// TIA Portal V16 export
// export: Created 2021-06-28T11:45:27.8781745Z, ExportSetting WithDefaults, DisplayName Totally Integrated Automation Portal, DisplayVersion V16 Update 4, DisplayName TIA Portal Version Control Interface, DisplayVersion V16 Update 2, DisplayName TIA Portal Openness, DisplayVersion V16 Update 4, DisplayName STEP 7 Professional, DisplayVersion V16 Update 4, DisplayName STEP 7 Safety, DisplayVersion V16, DisplayName WinCC Advanced, DisplayVersion V16 Update 4
FUNCTION "MQTT_MESSAGES_SEND" : Void   // FC10, FBD
{ S7_Optimized_Access := 'TRUE' }
VERSION : 0.1
// MQTT MESSAGES
// stored: AutoNumber true, IsIECCheckEnabled false, SetENOAutomatically false, UDAEnableTagReadback false
   VAR_TEMP
      TEMP0 : String;
      TEMP1 : String;
      TEMP3 : String;
      TEMP4 : String;
      TEMP5 : String;
      TEMP11 : String;
      wtemp1 : WString;
      wtemp2 : WString;
      wtemp3 : WString;
      wtemp4 : WString;
      TEMP6 : String;
      temp13 : String;
      temp14 : String;
      temp15 : String;
      wtemp14 : WString;
      wtemp16 : WString;
      temp110 : String;
      wtemp_null : WString;
      temp_rej1 : String;
      temp_rej2 : WString;
      TEMP : WString;
      TEMP_REJECT_TM_STMP : String;
      TEMP_BIT_BOOL1 : Bool;
   END_VAR
BEGIN

REGION Network 1 (SCL): Message_UID
   // MESSAGE_UID_FORMAT
   "MQTT_BLOCK".MSG_UID_data := CONCAT(IN1 := '"', IN2 :="MQTT_BLOCK".INDUCT_ID, IN3 := '_', IN4 := "MQTT_BLOCK".TIMESTAMP, IN5 := '"');
END_REGION

REGION Network 2 (SCL): CommonMessage
   // COMMON_MESSAGE
   "MQTT_BLOCK".COMMON_MESSAGE:=CONCAT(IN1:='{"message_uid":',IN2:="MQTT_BLOCK".MSG_UID_data,IN3:=',"induct_id":',IN4:="MQTT_BLOCK".INDUCT_ID,IN5:=',"timestamp":',
                                       IN6:="MQTT_BLOCK".TIMESTAMP,IN7:=',"data":{');
END_REGION

REGION Network 3 (SCL): ShipmentInfoMessage_ok_28.3.2021
   // // shipment INFO MQTT Message//
   IF "Info_Time_Mov_Bit" THEN
       #TEMP1 := CONCAT(IN1 := '{"message_uid":', IN2 := '"', IN3 := "MQTT_BLOCK".INDUCT_ID, IN4 := '_', IN5 := "MQTT_BLOCK".TimeStamp_Info, IN6 := '","induct_id":', IN7 := "MQTT_BLOCK".INDUCT_ID, IN8 := ',"timestamp":', IN9 := "MQTT_BLOCK".TimeStamp_Info, IN10 := ',"data":{"weight":', IN11 := "DATA_TCP".weight_string, IN12 := ',"barcodes":[');
       #TEMP3 := CONCAT(IN1 := '],"height":', IN2 := "DATA_TCP".STRING_H_INFO, IN3 := ',"length":', IN4 := "DATA_TCP".STRING_L_INFO, IN5 := ',"breadth":', IN6 := "DATA_TCP".STRING_B_INFO, IN7 := ',"weight_status_code":"',
                        IN8 := "MQTT_BLOCK".WEIGHT_STATUS_CODE, IN9 := '","vms_status_code":"', IN10 := "MQTT_BLOCK".VMS_STATUS_CODE, IN11 := '","scan_status_code":"',
                        IN12 := "MQTT_BLOCK".SCAN_STATUS_CODE, IN13 := '","uid":', IN14 := "MQTT_BLOCK".uid_1, IN15 := '');
       #wtemp1 := STRING_TO_WSTRING(#TEMP1);
       #wtemp4 := STRING_TO_WSTRING("DATA_TCP".String_To_String_Barcode);

       #wtemp2 := STRING_TO_WSTRING(#TEMP3);
       #wtemp3 := STRING_TO_WSTRING('}}');

       IF "DATA_TCP".STRING_L = '' THEN
           "DATA_TCP".STRING_L_INFO := '0';
       ELSE
           "DATA_TCP".STRING_L_INFO := "DATA_TCP".STRING_L;
       END_IF;

       IF "DATA_TCP".STRING_B = '' THEN
           "DATA_TCP".STRING_B_INFO := '0';
       ELSE
           "DATA_TCP".STRING_B_INFO := "DATA_TCP".STRING_B;
       END_IF;
       IF "DATA_TCP".STRING_H = '' THEN
           "DATA_TCP".STRING_H_INFO := '0';
       ELSE
           "DATA_TCP".STRING_H_INFO := "DATA_TCP".STRING_H;
       END_IF;


       IF "Aligner_Buffer_Module_Status" = 20 THEN
           "MQTT_BLOCK".MQTT_SHIPMENT_INFO := #wtemp_null;

       ELSIF "Aligner_Buffer_Module_Status" <> 20 & "Aligner_Buffer_Module_Status" < 300 THEN
           "MQTT_BLOCK".MQTT_SHIPMENT_INFO := CONCAT_WSTRING(IN1 := #wtemp1, IN2 := #wtemp4, IN3 := #wtemp2, IN4 := #wtemp3);
       END_IF;
       IF #wtemp4 = STRING_TO_WSTRING("DATA_TCP".String_To_String_Barcode) THEN
           "Trig_Info_CMD" := 1;
       END_IF;
       END_IF;
   // program end for shipment_info//
END_REGION

REGION Network 4 (SCL): HealthMessage WITH ERROR CODES
   // Induct Health MQTT Message
   IF "TIME_MOVE_HEALTH" & "ActualHealthStatus"=0 THEN
       IF "MQTT_BLOCK"."MQTT-OK" = 0 THEN "MQTT_BLOCK".health_induct_mqtt.message := '1'; "HEALTH_TR_2" := 1;
       ELSIF "Function_DB".IN_DWS_Alarm_DB = 0 THEN "MQTT_BLOCK".health_induct_mqtt.message := '403'; "HEALTH_TR_2" := 1;
       ELSIF "Function_DB".IN_Aligner_Alarm_DB  THEN "MQTT_BLOCK".health_induct_mqtt.message := '401'; "HEALTH_TR_2" := 1;
       ELSIF "Function_DB".IN_Barrier_Alarm_DB = 0 THEN "MQTT_BLOCK".health_induct_mqtt.message := '407'; "HEALTH_TR_2" := 1;
       ELSIF "Function_DB".IN_BUFFER_LEFT_ALARM_DB = 0 THEN "MQTT_BLOCK".health_induct_mqtt.message := '408'; "HEALTH_TR_2" := 1;
       ELSIF "Function_DB".IN_Buffer_Right_Alarm_DB = 0 THEN "MQTT_BLOCK".health_induct_mqtt.message := '409'; "HEALTH_TR_2" := 1;
       ELSIF "Error_Bit_Weight_Module"  THEN "MQTT_BLOCK".health_induct_mqtt.message := '410'; "HEALTH_TR_2" := 1;
       ELSIF "Error_Timeout"  THEN
           IF "IN_DWS_FAULT"  THEN
               "MQTT_BLOCK".health_induct_mqtt.message := '411';
               "HEALTH_TR_2" := 1;
           ELSIF "OUT_DWS_FAULT" THEN
               "MQTT_BLOCK".health_induct_mqtt.message := '412';
               "HEALTH_TR_2" := 1;
           ELSIF "DN_ALIGNER_FAULT" THEN
               "MQTT_BLOCK".health_induct_mqtt.message := '413';
               "HEALTH_TR_2" := 1;
           ELSIF "UP_ALIGNER_FAULT" THEN
               "MQTT_BLOCK".health_induct_mqtt.message := '414';
               "HEALTH_TR_2" := 1;
           ELSIF "IN_BUFFER_FAULT" THEN
               "MQTT_BLOCK".health_induct_mqtt.message := '415';
               "HEALTH_TR_2" := 1;
           ELSIF "OUT_BUFFER_FAULT" THEN
               "MQTT_BLOCK".health_induct_mqtt.message := '416';
               "HEALTH_TR_2" := 1;
           END_IF;

       ELSIF "IEC_Timer_0_DB_10".Q  THEN "MQTT_BLOCK".health_induct_mqtt.message := '100'; "HEALTH_TR_2" := 1;
       END_IF;
   ELSIF "ActualHealthStatus" &"TIME_MOVE_HEALTH" THEN "MQTT_BLOCK".health_induct_mqtt.message := ''; "HEALTH_TR_1" := 1;
   END_IF;

   #temp110 := CONCAT(IN1 := '{"message_uid":"',IN2:="MQTT_BLOCK".INDUCT_ID, IN3:='_', IN4:="MQTT_BLOCK".TimeStamp_Health , IN5:=' ","induct_id":', IN6:="MQTT_BLOCK".INDUCT_ID, IN7:=',"timestamp":', IN8:= "MQTT_BLOCK".TimeStamp_Health, IN9:=',"data":{"connected":', IN10 := "MQTT_BLOCK".health_induct_mqtt.connection, IN11 := ',"induct_healthy":', IN12 := "MQTT_BLOCK".health_induct_mqtt.induct_healthy,
                      IN13 := ',"error_code":"', IN14 := "MQTT_BLOCK".health_induct_mqtt.message, IN15 := '"}}');


   "MQTT_BLOCK".MQTT_INDUCT_HEALTH:=STRING_TO_WSTRING(#temp110);
END_REGION

REGION Network 5 (SCL): BotResponseMessage
   // BOT RESPONSE MQTT MESSAGE
   #temp13:= CONCAT(IN1 := '{"message_uid":', IN2:= '"',IN3:="MQTT_BLOCK".INDUCT_ID, IN4:='_', IN5:="MQTT_BLOCK".TimeStamp_Bot, IN6:='","induct_id":', IN7:="MQTT_BLOCK".INDUCT_ID,
                    IN8:=',"timestamp":', IN9:= "MQTT_BLOCK".TimeStamp_Bot, IN10:=',"data":{"bot_event":"going","response":',IN11:="MQTT_BLOCK".Bot_response.response,
                    IN12:=',"messages":"',IN13:="MQTT_BLOCK".Bot_response.message,IN14:='"}}');

   "MQTT_BLOCK".MQTT_BOT := STRING_TO_WSTRING(#temp13);

   IF "Buffer_Transfer_Seq_Status" < 20 & "MQTT_BLOCK".MQTT_BOT_GOING = 1 THEN
       "MQTT_BLOCK".Bot_response.response := 'true';
       "MQTT_BLOCK".MQTT_BOT_ARRIVED := 0;
   ELSIF "Buffer_Transfer_Seq_Status" >= 20 & "MQTT_BLOCK".MQTT_BOT_GOING = 1 THEN
       "MQTT_BLOCK".Bot_response.response := 'false';
       "MQTT_BLOCK".Bot_response.message := 'shipment_initiated_already';
   END_IF;
END_REGION

REGION Network 6 (SCL): ShipmentRejectionMessage
   // SHIPMENT REJECTION MQTT MESSAGE
   IF "REJ_TIME_BIT" & "Aligner_Buffer_Module_Status" = 520 OR "Aligner_Buffer_Module_Status" = 320 THEN

       "MQTT_BLOCK".uid_3 := "MQTT_BLOCK".uid;
       IF "Tag_76">15000 THEN
           "MQTT_BLOCK".WEIGHT_STATUS_CODE := '-1';
           END_IF;
       "MQTT_BLOCK".VMS_STATUS_CODE := '-1';

       IF "DATA_TCP".STRING_BARCODE = 'noread' OR "DATA_TCP".STRING_BARCODE = '' THEN
           "MQTT_BLOCK".SCAN_STATUS_CODE := '-1';
       END_IF;
       #temp_rej1 := CONCAT(IN1 := '{"message_uid":', IN2 := '"', IN3 := "MQTT_BLOCK".INDUCT_ID, IN4 := '_', IN5 := "MQTT_BLOCK".TimeStamp_Rejection, IN6 := '","induct_id":', IN7 := "MQTT_BLOCK".INDUCT_ID, IN8 := ',"timestamp":', IN9 := "MQTT_BLOCK".TimeStamp_Rejection, IN10 := ',"data":{"weight":', IN11 := "DATA_TCP".weight_string, IN12 := ',"barcodes":[');
       #TEMP3 := CONCAT(IN1 := '],"height":', IN2 := "DATA_TCP".STRING_H_INFO, IN3 := ',"length":', IN4 := "DATA_TCP".STRING_L_INFO, IN5 := ',"breadth":', IN6 := "DATA_TCP".STRING_B_INFO, IN7 := ',"weight_status_code":"',
                        IN8 := "MQTT_BLOCK".WEIGHT_STATUS_CODE, IN9 := '","vms_status_code":"', IN10 := "MQTT_BLOCK".VMS_STATUS_CODE, IN11 := '","scan_status_code":"',
                        IN12 := "MQTT_BLOCK".SCAN_STATUS_CODE, IN13 := '","uid":', IN14 := "MQTT_BLOCK".uid_3 , IN15 :='');
       #temp_rej2 := STRING_TO_WSTRING(#temp_rej1);
       #wtemp4 := STRING_TO_WSTRING("DATA_TCP".String_To_String_Barcode);
       #wtemp2 := STRING_TO_WSTRING(#TEMP3);
       #wtemp3 := STRING_TO_WSTRING('}}');

       "MQTT_BLOCK".MQTT_SHIPMENT_REJECTION := CONCAT_WSTRING(IN1 := #temp_rej2, IN2 := #wtemp4, IN3 := #wtemp2, IN4 := #wtemp3);
       "REJ_BIT_MSG" := 1;
   ELSE
       "MQTT_BLOCK".MQTT_SHIPMENT_REJECTION := STRING_TO_WSTRING('');
       "MQTT_BLOCK".WEIGHT_STATUS_CODE := '0';
       "MQTT_BLOCK".VMS_STATUS_CODE := '0';
       "MQTT_BLOCK".SCAN_STATUS_CODE := '0';
   END_IF;
END_REGION

REGION Network 7 (SCL): LAST_WILL_MESSAGE
   "MQTT_BLOCK".PARAMETER.willMessage :=CONCAT(IN1:='{"msgId":',IN2 :="MQTT_BLOCK".MSG_UID_data ,IN3:=',"inductId":1,"timestamp":',IN4:="MQTT_BLOCK".TIMESTAMP, IN5 := ',"data":{}}');
END_REGION
END_FUNCTION
